// TIA Portal V16 export
// export: Created 2019-09-22T13:16:38.230641Z, ExportSetting WithDefaults, DisplayName Totally Integrated Automation Portal, DisplayVersion V16, DisplayName TIA Portal Version Control Interface, DisplayVersion V16, DisplayName TIA Portal Openness, DisplayVersion V16, DisplayName STEP 7 Professional, DisplayVersion V16, DisplayName SIMATIC Energy Suite, DisplayVersion V16, DisplayName STEP 7 Safety, DisplayVersion V16, DisplayName WinCC Professional, DisplayVersion V16, DisplayName SIMATIC Visualization Architect, DisplayVersion V16
FUNCTION_BLOCK "LiftStartStop"   // FB2, FBD
{ S7_Optimized_Access := 'TRUE' }
VERSION : 0.1
// stored: AutoNumber true, IsIECCheckEnabled false, IsRetainMemResEnabled false, MemoryReserve 100, SetENOAutomatically false, UDAEnableTagReadback false
   VAR_INPUT
      autoStart : Bool;
      autoStop : Bool;
      plantOn : Bool;
      posCaseBelt : Int;
      lift1down : Bool;
      lift2down : Bool;
   END_VAR
   VAR_OUTPUT
      autoStarted : Bool;
      autoStopped : Bool;
   END_VAR
   VAR
      statCaseOnStopper : Bool;
      statAutoStopped : Bool;
   END_VAR
   VAR CONSTANT
      POS_STOPPER_1 : Int := 50;   // Position case stopper 1
      POS_STOPPER_2 : Int := 74;   // Position case stopper 2
      POS_STOPPER_3 : Int := 100;   // Position case stopper 3
   END_VAR
BEGIN

REGION Network 1
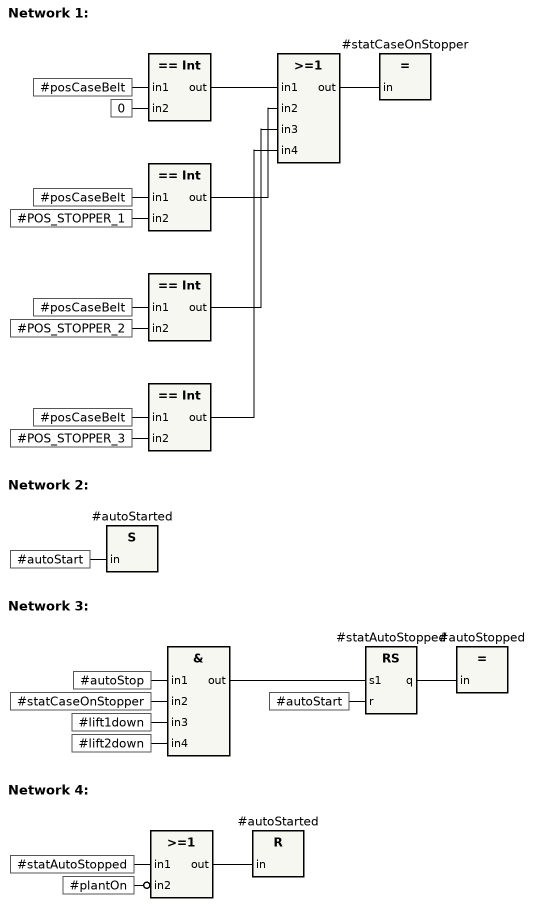
   #statCaseOnStopper := (#posCaseBelt = 0) OR (#posCaseBelt = #POS_STOPPER_1) OR (#posCaseBelt = #POS_STOPPER_2) OR (#posCaseBelt = #POS_STOPPER_3);
END_REGION

REGION Network 2
   IF #autoStart THEN #autoStarted := TRUE; END_IF;
END_REGION

REGION Network 3
   IF #autoStart THEN
       #statAutoStopped := FALSE;   // RS flip-flop
   END_IF;
   IF #autoStop AND #statCaseOnStopper AND #lift1down AND #lift2down THEN #statAutoStopped := TRUE; END_IF;
   #autoStopped := #statAutoStopped;
END_REGION

REGION Network 4
   IF #statAutoStopped OR NOT #plantOn THEN #autoStarted := FALSE; END_IF;
END_REGION
END_FUNCTION_BLOCK
